FUNCTION_BLOCK FB_Colleague IMPLEMENTS I_Colleague
VAR_INPUT
	iMediator : REFERENCE TO I_Mediator; // Mediator Interface
END_VAR

METHOD operation : BOOL
VAR_INPUT
	event : STRING;
END_VAR
IF __ISVALIDREF(iMediator) THEN
	iMediator.notify(THIS^,event);
END_IF
END_METHOD

END_FUNCTION_BLOCK

(* stored: Version 1.1.0.1, ProductVersion 3.1.4024.12
   POU FB_Colleague: Id {afb6d582-cdd4-4e93-9757-95f2ec75b624}, SpecialFunc None
   Method operation: Id {2a639bd1-c628-4980-8313-74cc776e7c0a} *)
